// TIA Portal V20 export
DATA_BLOCK "T5 EXCENTRIC"   // DB1118
{ S7_Optimized_Access := 'TRUE' }
AUTHOR : SAS
// stored: AutoNumber false, IsRetainMemResEnabled true, MemoryReserve 100, RetainMemoryReserve 100
   VAR RETAIN
      "Seq Status" : Struct
         ReadyToAuto : Bool;
         AutoON : Bool;
         WaitPiece : Bool;
         Stopped : Bool;
         "Step" : Struct
            Actual : Int;
            "-1" : Int;
            "-2" : Int;
            "-3" : Int;
            "-4" : Int;
            "-5" : Int;
            "-6" : Int;
            "-7" : Int;
            "-8" : Int;
            "-9" : Int;
            "Actual time" : Time_Of_Day;
            "-1 Time" : Time_Of_Day;
            "-2 Time" : Time_Of_Day;
            "-3 Time" : Time_Of_Day;
            "-4 Time" : Time_Of_Day;
            "-5 Time" : Time_Of_Day;
            "-6 Time" : Time_Of_Day;
            "-7 Time" : Time_Of_Day;
            "-8 Time" : Time_Of_Day;
            "-9 Time" : Time_Of_Day;
         END_STRUCT;
      END_STRUCT;
      Transitions : Struct
         Safe : Bool;   // Emergency
         Fault : Bool;   // Fault
         Auto : Bool;
         Manual : Bool;
         Pause : Bool;
         Stop : Bool;
         "Cycle start request" : Bool;
         "First Piece" : Bool;
         "Piece presence" : Bool;
         "Adjacent Machines" : Bool;   // Adjacent for start from initial position
         "Adjacent Machines Vertical" : Bool;   // Adjacent for start from vertical position
         Init_Sequence : Bool;
         "Movement conditions 1" : Bool;   // Pozitia 'Initial'
         "Movement conditions 2" : Bool;   // Pozitia 'Vertical'
         "Movement conditions 3" : Bool;
         "Movement conditions 4" : Bool;
         "Reset Fault" : Bool;
         "Bypass ilock" : Bool;
      END_STRUCT;
      Memory : Struct
         "Piece presence" : Bool;   // Cumulative piece presence
         "Piece absence" : Bool;   // No sensor triggered
         "Pipe Transfered" : Bool;   // Pipe transfered
         "Permanent Condition" : Bool;   // Permanent condition
         "Movement Fault" : Bool;   // Cumulative of Machine Fault condition
         "Local StopAuto" : Bool;   // Local StopAuto
         "Interlocks FW" : Bool;   // Interlocks for FORWARD
         "Interlocks BW" : Bool;   // Interlocks for BACKWARD
         FW_ON : Bool;   // Rotire 'Inainte'
         BW_ON : Bool;   // Rotire 'Inapoi'
         EX_AUTO_FW : Bool;   // Excentric Rotire 'Inainte' in Mod Automat
         FW_MANUAL : Bool;   // Rotire 'Inainte' in Mod Manual - Single Cycle Run
         OS_POSITION : Bool;   // OS NOTE POSITION
         EX_INITIAL : Bool;   // Pozitia 'Initial'
         EX_VERT : Bool;   // Pozitie 'Vertical'
         STEP_DONE_LANT : Bool;   // T5 Lant has done a Step
      END_STRUCT;
   END_VAR
BEGIN
END_DATA_BLOCK
